// TwinCAT 3 PLC project PushcorpCtrl
// ProgramVersion: 3.1.4023.0
// libraries:
//   Tc2_Standard, * (Beckhoff Automation GmbH)
//   Tc2_System, * (Beckhoff Automation GmbH)
//   Tc3_EventLogger, * (Beckhoff Automation GmbH)
//   Tc3_Module, * (Beckhoff Automation GmbH)
//   BASIC,3.31,OSCAT
//   Util,3.5.11.0,System
// project tree:
//   DUTs/DoDi/IO/ ST_DoDi.TcDUT, ST_DoDi_in.TcDUT, ST_DoDi_out.TcDUT
//   DUTs/FCU/ E_FCU_ControlMode.TcDUT, ST_FcuControl.TcDUT, ST_FcuControl_in.TcDUT, ST_FcuControl_out.TcDUT
//   DUTs/FCU/IO/ ST_FCUFLEX.TcDUT, ST_FCUFLEX_in.TcDUT, ST_FCUFLEX_in_bits.TcDUT, ST_FCUFLEX_out.TcDUT
//   DUTs/Motoman/IO/ ST_MotomanIO.TcDUT, ST_MotomanIO_in.TcDUT, ST_MotomanIO_out.TcDUT
//   DUTs/Motoman/ ST_MotomanCtrl.TcDUT, ST_MotomanCtrl_in.TcDUT, ST_MotomanCtrl_out.TcDUT
//   DUTs/OPCUA/ ST_OpcuaStatus.TcDUT, ST_OpcuaStatusError.TcDUT, ST_OpcuaStatus_in.TcDUT, ST_OpcuaStatus_out.TcDUT, U_OpcuaError.TcDUT
//   DUTs/SPINDLE/IO/ ST_Spindle.TcDUT, ST_Spindle_in.TcDUT, ST_Spindle_in_bits.TcDUT, ST_Spindle_out.TcDUT, ST_Spindle_out_bits.TcDUT
//   DUTs/SPINDLE/ ST_SpindleControl.TcDUT, ST_SpindleControl_in.TcDUT, ST_SpindleControl_out.TcDUT
//   DUTs/Testing/ ST_TestBasicControl.TcDUT, ST_TestBasicControl_in.TcDUT, ST_TestBasicControl_out.TcDUT, ST_TestBasicControl_sub1.TcDUT
//   GVLs/ GVL_io.TcGVL, GVL_opcua.TcGVL
//   / PlcTask.TcTTO
//   POUs/ FB_FCU.TcPOU, FB_Motoman.TcPOU, FB_HeartbeatMonitor.TcPOU, FB_Spindle.TcPOU, FB_TestBasic.TcPOU, MAIN.TcPOU, prgMotoman.TcPOU, PRG_OpcuaMonitor.TcPOU
// real-time tasks:
//   TASK PlcTask: cycle T#1ms, priority 20, ADS port 350
//   TASK Task EthIp: cycle T#1ms, priority 1, ADS port 301
// I/O:
//   DEVICE Device 1 (EtherCAT), AmsNetId 192.168.125.39.2.1
//     Term 1 (EK1200) [EK1200-5000 EtherCAT Power supply (2A E-Bus)]
//       Term 2 (EL6070-0033) [EL6070-0033 1Ch. Licence key terminal, individual licences]
//       Term 3 (EL1008) [EL1008 8Ch. Dig. Input 24V, 3ms]
//       Term 4 (EL2008) [EL2008 8Ch. Dig. Output 24V, 0.5A]
//       Term 5 (EK1110) [EK1110 EtherCAT extension]
//   DEVICE Device 2 (TC3 EIP Scanner), AmsNetId 192.168.125.39.3.1
//     FCU (EtherNet/IP Slave (generic)) // <INFO> </INFO> <EDS> C:\TwinCAT\3.1\Config\Io\EtherNetIP\ </EDS>
//     Spindle (EtherNet/IP Slave (generic)) // <INFO> </INFO> <EDS> C:\TwinCAT\3.1\Config\Io\EtherNetIP\ </EDS>
//     DX200 EtherNet/IP(TM) Module // <INFO> 192.168.1.20, DX200 EtherNet/IP(TM) Module (ProdCode: 1281, Rev: 1.01, Mac: 00:26:73:d2:4a:d9) </INFO> <EDS> C:\TwinCAT\3.1\Config\Io\EtherNetIP\ </EDS>
// variable links:
//   PushcorpCtrl/PushcorpCtrl Instance <-> Device 1 (EtherCAT)/Term 1 (EK1200)/Term 3 (EL1008)
//     PlcTask Inputs/GVL_io.DI0 <-> Channel 1/GVL_io.DI0
//   PushcorpCtrl/PushcorpCtrl Instance <-> Device 1 (EtherCAT)/Term 1 (EK1200)/Term 4 (EL2008)
//     PlcTask Outputs/GVL_io.DO0 <-> Channel 1/GVL_io.DO0
//   PushcorpCtrl/PushcorpCtrl Instance <-> Device 2 (TC3 EIP Scanner)/DX200 EtherNet/IP(TM) Module
//     PlcTask Inputs/GVL_io.Motoman_Full.in/data <-> DX200 IO/Inputs/DX200_in
//     PlcTask Outputs/GVL_io.Motoman_Full.out <-> DX200 IO/Outputs/DX200_out
//   PushcorpCtrl/PushcorpCtrl Instance <-> Device 2 (TC3 EIP Scanner)/FCU (EtherNet/IP Slave (generic))
//     PlcTask Inputs/GVL_io.FCU_Full.DevState <-> Inputs/GVL_io.FCU_Full.DevState
//     PlcTask Inputs/GVL_io.FCU_Full.in <-> FCU IO/Inputs/GVL_io.FCU_Full.in
//     PlcTask Outputs/GVL_io.FCU_Full.out <-> FCU IO/Outputs/GVL_io.FCU_Full.out
//   PushcorpCtrl/PushcorpCtrl Instance <-> Device 2 (TC3 EIP Scanner)/Spindle (EtherNet/IP Slave (generic))
//     PlcTask Inputs/GVL_io.Spindle_Full.DevState <-> Inputs/GVL_io.Spindle_Full.DevState
//     PlcTask Inputs/GVL_io.Spindle_Full.in <-> Spindle IO/Inputs/GVL_io.Spindle_Full.in
//     PlcTask Outputs/GVL_io.Spindle_Full.out <-> Spindle IO/Outputs/GVL_io.Spindle_Full.out

CONFIGURATION PushcorpCtrl
    RESOURCE PLC ON TwinCAT3
        TASK PlcTask(INTERVAL := T#1ms, PRIORITY := 20);
        PROGRAM MAIN WITH PlcTask : MAIN;
    END_RESOURCE
END_CONFIGURATION

// ---- DUTs/DoDi/IO/ST_DoDi.TcDUT
TYPE ST_DoDi :
STRUCT	
	input	: ST_DoDi_in;	
	
	output	: ST_DoDi_out;	
END_STRUCT
END_TYPE

// ---- DUTs/DoDi/IO/ST_DoDi_in.TcDUT
TYPE ST_DoDi_in :
STRUCT
	DI0	AT %I*	: BOOL;
END_STRUCT
END_TYPE

// ---- DUTs/DoDi/IO/ST_DoDi_out.TcDUT
TYPE ST_DoDi_out :
STRUCT
	DO0	AT %Q*	: BOOL;
END_STRUCT
END_TYPE

// ---- DUTs/FCU/E_FCU_ControlMode.TcDUT
{attribute 'qualified_only'}
{attribute 'strict'}
TYPE E_FCU_ControlMode :
(
	Position := 0,
	Force := 1,
	SoftTouch := 3
) WORD;
END_TYPE

// ---- DUTs/FCU/IO/ST_FCUFLEX.TcDUT
{attribute 'pack_mode' := '2'}
TYPE ST_FCUFLEX :
STRUCT
	DevState AT %I* : UINT;
		
	in AT %I* : ST_FCUFLEX_in;
		
	out AT %Q* : ST_FCUFLEX_out;
END_STRUCT
END_TYPE

// ---- DUTs/FCU/IO/ST_FCUFLEX_in.TcDUT
{attribute 'pack_mode' := '2'}
TYPE ST_FCUFLEX_in :
STRUCT
	Flags : ST_FCUFLEX_in_bits;
	ActForce : INT;
	ActPos : WORD;
	AccelGravity : INT;
	CommandForce : INT;
	CommandPos : WORD;
	PayloadWeigth : WORD;
	ControlMode : WORD;
	MaxForce : WORD;
	MaxPos : WORD;
END_STRUCT
END_TYPE

// ---- DUTs/FCU/IO/ST_FCUFLEX_in_bits.TcDUT
TYPE ST_FCUFLEX_in_bits :
STRUCT
	hb : BIT;
	Hostcomm : BIT;
	ToolComm : BIT;
	MetricUnits : BIT;
	PosLimit : BIT;
	NegLimit : BIT;
	AtWeightPosition : BIT;
	WeighInProgress : BIT;
	WeightValid : BIT;
	 {attribute 'hide'}
	_reserved1 : BIT;
	 {attribute 'hide'}
	_reserved2 : BIT;
	 {attribute 'hide'}
	_reserved3 : BIT;
	 {attribute 'hide'}
	_reserved4 : BIT;
	 {attribute 'hide'}
	_reserved5 : BIT;
	 {attribute 'hide'}
	_reserved6 : BIT;
	 {attribute 'hide'}
	_reserved7 : BIT;
END_STRUCT
END_TYPE

// ---- DUTs/FCU/IO/ST_FCUFLEX_out.TcDUT
{attribute 'pack_mode' := '2'}
TYPE ST_FCUFLEX_out :
STRUCT
	CommandForce : INT;
	CommandPosition : WORD;
	PayloadWeight : WORD;
	ControlMode : WORD := 3;	// SoftTouch
	WeighPayloadNow : WORD;
END_STRUCT
END_TYPE

// ---- DUTs/FCU/ST_FcuControl.TcDUT
TYPE ST_FcuControl :
STRUCT
	status	: ST_OpcuaStatus;
	
	input	: ST_FcuControl_in;	
	
	{attribute 'OPC.UA.DA.Access' := '1'}
	output	: ST_FcuControl_out;
END_STRUCT
END_TYPE

// ---- DUTs/FCU/ST_FcuControl_in.TcDUT
{attribute 'OPC.UA.DA.StructuredType' := '1'}
TYPE ST_FcuControl_in :
STRUCT
	SetForce	: REAL;
	SetPosition	: REAL;
	SetWeight	: REAL;
	SetControlMode	: E_FCU_ControlMode := E_FCU_ControlMode.SoftTouch;
	WeighPayloadNow	: BOOL;
END_STRUCT
END_TYPE

// ---- DUTs/FCU/ST_FcuControl_out.TcDUT
{attribute 'OPC.UA.DA.StructuredType' := '1'}
TYPE ST_FcuControl_out :
STRUCT
	ActForce	: REAL;
	ActPos	: REAL;
	ActWeight	: REAL;
	Contact	: BOOL;
	WeightValid : BOOL;	
	Error	: UINT;
END_STRUCT
END_TYPE

// ---- DUTs/Motoman/IO/ST_MotomanIO.TcDUT
TYPE ST_MotomanIO :
STRUCT
	DevState AT %I* : UINT;
		
	in AT %I* : ST_MotomanIO_in;
		
	out AT %Q* : ST_MotomanIO_out;
END_STRUCT
END_TYPE

// ---- DUTs/Motoman/IO/ST_MotomanIO_in.TcDUT
TYPE ST_MotomanIO_in :
STRUCT
	data	: ARRAY[0..63] OF BYTE;
END_STRUCT
END_TYPE

// ---- DUTs/Motoman/IO/ST_MotomanIO_out.TcDUT
TYPE ST_MotomanIO_out :
STRUCT
	Cmd	: WORD;
	Vals	: ARRAY[0..5] OF WORD;
	Reserved	: ARRAY[0..49] OF BYTE;
END_STRUCT
END_TYPE

// ---- DUTs/Motoman/ST_MotomanCtrl.TcDUT
TYPE ST_MotomanCtrl :
STRUCT
	status	: ST_OpcuaStatus;
	
	input	: ST_MotomanCtrl_in;	
	
	{attribute 'OPC.UA.DA.Access' := '1'}
	output	: ST_MotomanCtrl_out;
END_STRUCT
END_TYPE

// ---- DUTs/Motoman/ST_MotomanCtrl_in.TcDUT
TYPE ST_MotomanCtrl_in :
STRUCT
	EnableJoystick	: BOOL;
	Value_1	: REAL;
	Value_2	: REAL;
	Value_3	: REAL;
	Value_4	: REAL;
	Value_5	: REAL;
	Value_6	: REAL;
END_STRUCT
END_TYPE

// ---- DUTs/Motoman/ST_MotomanCtrl_out.TcDUT
{attribute 'OPC.UA.DA.StructuredType' := '1'}
TYPE ST_MotomanCtrl_out :
STRUCT	
	Error	: UINT;
END_STRUCT
END_TYPE

// ---- DUTs/OPCUA/ST_OpcuaStatus.TcDUT
TYPE ST_OpcuaStatus :
STRUCT
	input	: ST_OpcuaStatus_in;
	
	{attribute 'OPC.UA.DA.Access' := '1'}
	output	: ST_OpcuaStatus_out;
END_STRUCT
END_TYPE

// ---- DUTs/OPCUA/ST_OpcuaStatusError.TcDUT
TYPE ST_OpcuaStatusError :
STRUCT
	DevDisconnected	: BIT;
	ClientHbLost	: BIT;
END_STRUCT
END_TYPE

// ---- DUTs/OPCUA/ST_OpcuaStatus_in.TcDUT
TYPE ST_OpcuaStatus_in :
STRUCT
	Heartbeat	: BOOL;
END_STRUCT
END_TYPE

// ---- DUTs/OPCUA/ST_OpcuaStatus_out.TcDUT
TYPE ST_OpcuaStatus_out :
STRUCT
	Heartbeat	: BOOL;
	Error	: UINT;	// 0 = No error
	Connected	: BOOL;
END_STRUCT
END_TYPE

// ---- DUTs/OPCUA/U_OpcuaError.TcDUT
TYPE U_OpcuaError :
UNION
	Value	: UINT;
	Bits	: ST_OpcuaStatusError;
END_UNION
END_TYPE

// ---- DUTs/SPINDLE/IO/ST_Spindle.TcDUT
{attribute 'pack_mode' := '2'}
TYPE ST_Spindle :
STRUCT
	DevState AT %I*	: UINT;
	in AT %I*	: ST_Spindle_in;
	out	 AT %Q* : ST_Spindle_out;
END_STRUCT
END_TYPE

// ---- DUTs/SPINDLE/IO/ST_Spindle_in.TcDUT
TYPE ST_Spindle_in :
STRUCT
	flags	: ST_Spindle_in_bits;
	SpindleSpeed	: INT;
	MotorLoad	: INT;
END_STRUCT
END_TYPE

// ---- DUTs/SPINDLE/IO/ST_Spindle_in_bits.TcDUT
{attribute 'pack_mode' := '2'}
TYPE ST_Spindle_in_bits :
STRUCT
	Contactor1	: BIT;
	Contactor2	: BIT;
	DriveError	: BIT;
	RpmLT5		: BIT;	
	DI5			: BIT;
	DI6			: BIT;
	DI7			: BIT;
	DI8			: BIT;
	Reserved	: BIT;	// Force 2 bytes, probably not needed
END_STRUCT
END_TYPE

// ---- DUTs/SPINDLE/IO/ST_Spindle_out.TcDUT
TYPE ST_Spindle_out :
STRUCT
	flags	: ST_Spindle_out_bits;
	SpindleSpeed	: INT;
	Reserved	: INT;
END_STRUCT
END_TYPE

// ---- DUTs/SPINDLE/IO/ST_Spindle_out_bits.TcDUT
{attribute 'pack_mode' := '2'}
TYPE ST_Spindle_out_bits :
STRUCT
	ServoEnable	: BIT;
	ResetFault	: BIT;
	DO3	: BIT;
	DO4	: BIT;
	DO5	: BIT;
	DO6	: BIT;
	DO7	: BIT;
	DO8	: BIT;	
	Reserved	: BIT;	// Force 2 bytes, probably not needed
END_STRUCT
END_TYPE

// ---- DUTs/SPINDLE/ST_SpindleControl.TcDUT
{attribute 'OPC.UA.DA.StructuredType' := '1'}
TYPE ST_SpindleControl :
STRUCT
	status	: ST_OpcuaStatus;
	
	input	: ST_SpindleControl_in;
	
	{attribute 'OPC.UA.DA.Access' := '1'}
	output	: ST_SpindleControl_out;
END_STRUCT
END_TYPE

// ---- DUTs/SPINDLE/ST_SpindleControl_in.TcDUT
{attribute 'OPC.UA.DA.StructuredType' := '1'}
TYPE ST_SpindleControl_in :
STRUCT
	Execute	: BOOL;
	(*{attribute 'OPC.UA.DA.AnalogItemType' := '1'}
	{attribute 'OPC.UA.DA.AnalogItemType.EngineeringUnits' := '5059638'}
	{attribute 'OPC.UA.DA.AnalogItemType.EURange' := '-15000.0:15000.0'}
	{attribute 'OPC.UA.DA.AnalogItemType.WriteBehavior' := '1'}*)
	SetVelo	: REAL;
END_STRUCT
END_TYPE

// ---- DUTs/SPINDLE/ST_SpindleControl_out.TcDUT

TYPE ST_SpindleControl_out :
STRUCT
	ActVelo	: REAL;	//Speed in RPMs
	Ready	: BOOL;
	Error	: UINT;	// 0 = No error
END_STRUCT
END_TYPE

// ---- DUTs/Testing/ST_TestBasicControl.TcDUT
TYPE ST_TestBasicControl :
STRUCT
	status	: ST_OpcuaStatus;	
	input	: ST_TestBasicControl_in;	
	
	{attribute 'OPC.UA.DA.Access' := '1'}
	output	: ST_TestBasicControl_out;
END_STRUCT
END_TYPE

// ---- DUTs/Testing/ST_TestBasicControl_in.TcDUT
TYPE ST_TestBasicControl_in :
STRUCT
	arrTest	: ARRAY[0..10] OF DINT;
	DO0	: BOOL;
	in1	: DINT;
	int2	: DINT;
	stSub1In	: ST_TestBasicControl_sub1; 
	inStr1	: STRING(255);	
END_STRUCT
END_TYPE

// ---- DUTs/Testing/ST_TestBasicControl_out.TcDUT
TYPE ST_TestBasicControl_out :
STRUCT
	DI0	: BOOL;
	out1	: DINT;
	out2	: DINT;
	stSub1Out	: ST_TestBasicControl_sub1;
	outStr1	: STRING(255);
	arrTest	: ARRAY[0..1] OF BYTE;
END_STRUCT
END_TYPE

// ---- DUTs/Testing/ST_TestBasicControl_sub1.TcDUT
TYPE ST_TestBasicControl_sub1 :
STRUCT
	sub1val	: DINT;
END_STRUCT
END_TYPE

// ---- GVLs/GVL_io.TcGVL
{attribute 'qualified_only'}
VAR_GLOBAL
	DI0 AT %I*	: BOOL;
	DO0 AT %Q*	: BOOL;
	
	Spindle_Full	: ST_Spindle;
	FCU_Full	: ST_FCUFLEX;
	
	
	DX200_in AT %I*	: ARRAY [0..7] OF BYTE;
	DX200_out AT %Q*	: ARRAY [0..7] OF BYTE;
	
	Motoman_Full	: ST_MotomanIO;
END_VAR

// ---- GVLs/GVL_opcua.TcGVL
{attribute 'qualified_only'}
VAR_GLOBAL
	{attribute 'OPC.UA.DA' := '1'}	
	stFcuControl	: ST_FcuControl;
	
	{attribute 'OPC.UA.DA' := '1'}
	stSpindleControl	: ST_SpindleControl;
	
	{attribute 'OPC.UA.DA' := '1'}	
	stTestBasic	: ST_TestBasicControl;
	
	{attribute 'OPC.UA.DA' := '1'}	
	stMotomanControl	: ST_MotomanCtrl;
END_VAR

// ---- POUs/MAIN.TcPOU
PROGRAM MAIN
VAR
	fbSpindle	: FB_Spindle;
	fbFcu	: FB_FCU;
	fbMotoman	: FB_Motoman;
	
	
	spin: REFERENCE TO ST_SpindleControl;
	fcu: REFERENCE TO ST_FcuControl;
	
	motoman	: REFERENCE TO ST_MotomanCtrl;
	motomanErr: BOOL;
END_VAR

//prgMotoman();

// Set ref vars for convenience of shorter names 
spin REF= GVL_opcua.stSpindleControl;
fcu REF=GVL_opcua.stFcuControl;
motoman REF= GVL_opcua.stMotomanControl;

// Monitor opcua heartbeat data in a Method for convenience.  This can be easily ignored if calling the FB without opcua 
fbSpindle.OpcuaMonitor(OpcuaData:= spin, Error=> );
fbSpindle(
	Enable:= spin.input.Execute, 
	SetVelo:= spin.input.SetVelo, 
	data:= GVL_io.Spindle_Full, 
	ActVelo=> spin.output.ActVelo, 
	Ready=> spin.output.Ready, 
	Error=> spin.output.Error);


fbFcu.OpcuaMonitor(OpcuaData:= fcu, Error=> );
fbFcu(
	SetForce:= fcu.input.SetForce, 
	SetPosition:= fcu.input.SetPosition, 
	SetWeight:= fcu.input.SetWeight, 
	SetControlMode:= fcu.input.SetControlMode, 
	WeightPayload:= fcu.input.WeighPayloadNow, 
	data:= gvl_io.FCU_Full, 
	ActForce=> fcu.output.ActForce, 
	ActPos=> fcu.output.ActPos, 
	ActWeight=> fcu.output.ActWeight,
	Contact=> fcu.output.Contact,
	WeightValid=> fcu.output.WeightValid, 
	Error=> fcu.output.Error);
	
fbMotoman.OpcuaMonitor(OpcuaData:= GVL_opcua.stMotomanControl, Error=> motomanErr);
fbMotoman(
	EnableJoystick:= NOT motomanErr, 
	Value_1:= motoman.input.Value_1, 
	Value_2:= motoman.input.Value_2, 
	Value_3:= motoman.input.Value_3, 
	Value_4:= , 
	Value_5:= , 
	Value_6:= , 
	data:= GVL_io.Motoman_Full, 
	Error=> );
	
// DI0 := DO0, for testing
GVL_io.DO0 := GVL_opcua.stTestBasic.input.DO0;
GVL_opcua.stTestBasic.output.DI0 := GVL_io.DI0;

END_PROGRAM

// ---- POUs/FB_Spindle.TcPOU
FUNCTION_BLOCK FB_Spindle
VAR_INPUT
	Enable	: BOOL; // Enable the servo
	SetVelo	: REAL;	// Speed in RPMs
END_VAR
VAR_IN_OUT
	data	: ST_Spindle;	// Ethernet IP data
END_VAR
VAR_OUTPUT
	ActVelo	: REAL;	//Speed in RPMs
	Ready	: BOOL; // Servo ready to move
	Error	: UINT; // 0 = OK, 1 = not connected
END_VAR
VAR
	rTargetVel	: REAL;	
	fbTrigEnable	: BOOL;	
	iState	: DINT;	
	fbDelay	: TON;
	bRunDelay	: BOOL;
	uiDevState: UINT;
END_VAR

IF NOT Enable THEN
	iState := 0;
END_IF

uiDevState := data.DevState;

// Scale target rpm
rTargetVel := SCALE_R(
				X:= SetVelo, 
				I_LO:= -15000, 
				I_HI:= 15000, 
				O_LO:= -30000, 
				O_HI:= 30000);
				
fbDelay(IN:= bRunDelay, PT:= T#1000MS, Q=> , ET=> );				

CASE iState OF
0:	// Default, set all output to 0
	MEMSET(ADR(data.out.flags), 0, SIZEOF(data.out.flags));
	bRunDelay := FALSE;
	IF Enable THEN
		iState := 10;
	END_IF
10:
	IF data.in.flags.DriveError THEN
		data.out.flags.ResetFault := TRUE;
		iState := 20;	// Reset state
	ELSE			
		iState := 100;	// OK to run
	END_IF	
20:
	data.out.flags.ServoEnable := FALSE;
	data.out.flags.ResetFault := data.in.flags.DriveError;
	bRunDelay := TRUE;	// Don't try to power on for at least a second
	IF NOT data.in.flags.DriveError AND fbDelay.Q THEN
		iState := 100;
		bRunDelay := FALSE;
	END_IF
	
100:
	data.out.flags.ServoEnable := TRUE;
	data.out.SpindleSpeed := TO_INT(rTargetVel);
	
	IF data.in.flags.DriveError THEN
		iState := 999;
	END_IF
	
999: // Stay in fault state until error can be examined
	data.out.flags.ServoEnable := FALSE;
	;
END_CASE


Error := TO_UINT(data.in.flags.DriveError);
Ready := Error = 0 AND data.in.flags.Contactor1 AND data.in.flags.Contactor2 AND data.DevState = 0;


IF data.in.flags.RpmLT5 THEN
	ActVelo := 0;
ELSE
	ActVelo := SCALE_R(
		X:= data.in.SpindleSpeed, 
		I_LO:= -30000, 
		I_HI:= 30000, 
		O_LO:= -15000, 
		O_HI:= 15000);
END_IF

METHOD OpcuaMonitor : BOOL
VAR_INPUT
END_VAR
VAR_IN_OUT
	OpcuaData	: ST_SpindleControl;
END_VAR
VAR_OUTPUT
	Error	: BOOL;
END_VAR
VAR_INST
	fbHbMonitor	: FB_HeartbeatMonitor;
	fbBlink	: BLINK;
END_VAR
fbHbMonitor(IN:= OpcuaData.status.input.Heartbeat, PT:= T#2.5S, Q=> );

IF NOT fbHbMonitor.Q THEN
	MEMSET(ADR(OpcuaData.input), 0, SIZEOF(OpcuaData.input));
	Error := TRUE;
ELSE
	Error := FALSE;
END_IF

fbBlink(ENABLE:= TRUE, TIMELOW:= T#500MS, TIMEHIGH:= T#500MS, OUT=> OpcuaData.status.output.Heartbeat);
OpcuaData.status.output.Connected := (THIS^.uiDevState = 0);
END_METHOD

END_FUNCTION_BLOCK

// ---- POUs/FB_HeartbeatMonitor.TcPOU
FUNCTION_BLOCK FB_HeartbeatMonitor
VAR_INPUT
	IN	: BOOL;
	PT	: TIME := T#2S;
END_VAR
VAR_OUTPUT
	Q	: BOOL;
END_VAR
VAR
	fbHbTimeout: TON;
	bLastHB: BOOL;
END_VAR

fbHbTimeout(IN:= (bLastHB = IN), PT:= PT, Q=> Q, ET=> );
Q := NOT fbHbTimeout.Q;
bLastHB := IN;

END_FUNCTION_BLOCK

// ---- POUs/FB_FCU.TcPOU
FUNCTION_BLOCK FB_FCU
VAR_INPUT
	SetForce	: REAL;	// Desired force in NM
	SetPosition	: REAL;	// Desired position in mm
	SetWeight	: REAL;	// Manually specify the weight, leave 0 if using WeightPayload
	SetControlMode	: E_FCU_ControlMode := E_FCU_ControlMode.Force;	// Position, Force, Soft Touch
	WeightPayload	: BOOL;	// Weight the payload now
END_VAR
VAR_IN_OUT
	data	: ST_FCUFLEX;	// Raw data from Ethernet/IP
END_VAR
VAR_OUTPUT
	ActForce	: REAL;	// Actual force in NM
	ActPos	: REAL;	// Actual position in mm
	ActWeight	: REAL;	// Actual weight in KG
	Contact	: BOOL;	// Contact state
	WeightValid : BOOL; // Is the weight valid or not initialized
	Error	: UINT;	// 
END_VAR
VAR
	bLastHB	: BOOL;
	bOk	: BOOL;	
	fbHbTimeout	: TON;
	
	rScaledForce: REAL;
	rTemp	: REAL;	
	rMaxPos	: REAL;
	uiDevState: UINT;
END_VAR

uiDevState := data.DevState;
// Check comms and heartbeat
bOk := TRUE;	
fbHbTimeout(IN:= (bLastHB = data.in.Flags.hb), PT:= T#2S, Q=> , ET=> );
bLastHB := data.in.Flags.hb;
	
IF fbHbTimeout.Q OR NOT data.in.Flags.Hostcomm OR NOT data.in.Flags.ToolComm THEN
	bOk := FALSE;
END_IF

// Scale data from FCU
ActForce := data.in.ActForce / 10.0;
ActPos := data.in.ActPos / 100.0;
ActWeight := data.in.PayloadWeigth / 100.0;
// Determine contact
rMaxPos := data.in.MaxPos  / 100.0;
Contact := (ActPos >= 2.0 AND ActPos <= rMaxPos - 2.0);
WeightValid := data.in.Flags.WeightValid;

// Scale and write data to FCU
data.out.ControlMode := TO_WORD(SetControlMode);
data.out.CommandForce := TO_INT(SetForce * 10.0);
data.out.CommandPosition := TO_WORD(SetPosition * 100.0);
data.out.PayloadWeight := TO_WORD(SetWeight * 100.0);
data.out.WeighPayloadNow := TO_WORD(WeightPayload);



Error := TO_UINT(NOT bOk);

METHOD OpcuaMonitor : BOOL
VAR_INPUT
END_VAR
VAR_IN_OUT
	OpcuaData	: ST_FcuControl;
END_VAR
VAR_OUTPUT
	Error	: BOOL;
END_VAR
VAR_INST
	fbHbMonitor	: FB_HeartbeatMonitor;
	fbBlink	: BLINK;	
	err	: U_OpcuaError;
END_VAR
fbHbMonitor(IN:= OpcuaData.status.input.Heartbeat, PT:= T#2.5S, Q=> );
err.Value := 0;
IF NOT fbHbMonitor.Q THEN
	// There's no way to simply disable the fcu and it defaults to position mode.  Trying to move to position 0
	// will cause a significant force
	OpcuaData.input.SetControlMode := E_FCU_ControlMode.SoftTouch;
	OpcuaData.input.SetForce := 0;
	OpcuaData.input.WeighPayloadNow := FALSE;
	
	err.Bits.ClientHbLost := TRUE;
END_IF

OpcuaData.status.output.Connected := (THIS^.uiDevState = 0);
IF NOT OpcuaData.status.output.Connected THEN	// higher priority
	err.Bits.DevDisconnected := TRUE;	
END_IF

Error := err.Value <> 0;
OpcuaData.status.output.Error := err.Value;

fbBlink(ENABLE:= TRUE, TIMELOW:= T#500MS, TIMEHIGH:= T#500MS, OUT=> OpcuaData.status.output.Heartbeat);
END_METHOD

END_FUNCTION_BLOCK

// ---- POUs/FB_Motoman.TcPOU
FUNCTION_BLOCK FB_Motoman
VAR_INPUT
	EnableJoystick	: BOOL;
	Value_1	: REAL;
	Value_2	: REAL;
	Value_3	: REAL;
	Value_4	: REAL;
	Value_5	: REAL;
	Value_6	: REAL;	
END_VAR
VAR_IN_OUT
	data	: ST_MotomanIO;	// Raw data from Ethernet/IP
END_VAR
VAR_OUTPUT	
	Error	: UINT;	// 
END_VAR
VAR
	uiDevState: UINT;
	bOk	: BOOL;	
	fbHbTimeout	: TON;
	
	rMaxOutVel : REAL := 1000;

	
	
	pInt	: POINTER TO INT;
	pWord	: POINTER TO WORD;
END_VAR

uiDevState := data.DevState;
// Check comms and heartbeat
bOk := TRUE;	


(*valTemp := LIMIT(-0.6, Value_1, 0.6);

tempLin := F_LIN2(
	X:= valTemp, 
	X1:= -0.6, 
	Y1:= -1000, 
	X2:= 0.6, 
	Y2:= 1000);
	
tempInt := TO_INT(tempLin);

MEMMOVE(ADR(data.out.Vals[0]), ADR(tempInt), 2);
//data.out.Vals[0] := tempInt;
*)

data.out.Vals[0] := PrepareValue(Value_1, rMaxOutVel);
data.out.Vals[1] := PrepareValue(Value_2, rMaxOutVel);
data.out.Vals[2] := PrepareValue(Value_3, rMaxOutVel);

data.out.Cmd.0 := EnableJoystick;

data.out.Cmd.1 := data.out.Vals[0] <> 0 OR data.out.Vals[1] <> 0 OR data.out.Vals[2] <> 0;

IF NOT EnableJoystick THEN 
	MEMSET(ADR(data.out.Cmd), 0, SIZEOF(data.out.Cmd));
	MEMSET(ADR(data.out.Vals), 0, SIZEOF(data.out.Vals));
END_IF
Error := TO_UINT(NOT bOk);

METHOD OpcuaMonitor : BOOL
VAR_INPUT
END_VAR
VAR_IN_OUT
	OpcuaData	: ST_MotomanCtrl;
END_VAR
VAR_OUTPUT
	Error	: BOOL;
END_VAR
VAR_INST
	fbHbMonitor	: FB_HeartbeatMonitor;
	fbBlink	: BLINK;	
	err	: U_OpcuaError;
END_VAR
fbHbMonitor(IN:= OpcuaData.status.input.Heartbeat, PT:= T#2.5S, Q=> );

IF NOT fbHbMonitor.Q THEN
	MEMSET(ADR(OpcuaData.input), 0, SIZEOF(OpcuaData.input));
	Error := TRUE;
ELSE
	Error := FALSE;
END_IF

fbBlink(ENABLE:= TRUE, TIMELOW:= T#500MS, TIMEHIGH:= T#500MS, OUT=> OpcuaData.status.output.Heartbeat);
OpcuaData.status.output.Connected := (THIS^.uiDevState = 0);
END_METHOD

METHOD PrepareValue : INT
VAR_INPUT
	SetVal	: REAL;
	MaxOut	: REAL := 1000;
END_VAR
VAR
	tempWord: WORD;
	tempInt	: INT;
	valTemp: REAL;
	tempLin: REAL;
END_VAR
valTemp := LIMIT(-0.6, SetVal, 0.6);

tempLin := F_LIN2(
	X:= valTemp, 
	X1:= -0.6, 
	Y1:= -MaxOut, 
	X2:= 0.6, 
	Y2:= MaxOut);
	
tempInt := TO_INT(tempLin);

MEMMOVE(ADR(PrepareValue), ADR(tempInt), 2);
END_METHOD

END_FUNCTION_BLOCK

// ---- POUs/FB_TestBasic.TcPOU
FUNCTION_BLOCK FB_TestBasic
VAR_INPUT
	DO0	: BOOL; // Enable the servo	
END_VAR
VAR_IN_OUT
	data	: ST_TestBasic;	// Ethernet IP data
END_VAR
VAR_OUTPUT
	DI0	: BOOL;
	Ready	: BOOL;
	Error	: UINT; 
END_VAR
VAR
END_VAR

METHOD OpcuaMonitor : BOOL
VAR_INPUT
END_VAR
VAR_IN_OUT
	Data	: ST_SpindleControl;
END_VAR
VAR_OUTPUT
	Error	: BOOL;
END_VAR
VAR_INST
	fbHbMonitor	: FB_HeartbeatMonitor;
END_VAR
fbHbMonitor(IN:= Data.status.input.Heartbeat, PT:= T#2.5S, Q=> );

IF NOT fbHbMonitor.Q THEN
	MEMSET(ADR(Data.input), 0, SIZEOF(Data.input));
	Error := TRUE;
ELSE
	Error := FALSE;
END_IF
END_METHOD

END_FUNCTION_BLOCK

// ---- POUs/prgMotoman.TcPOU
PROGRAM prgMotoman
VAR
	pReal	: POINTER TO REAL;
	rVal	: REAL;
	
	pInt	: POINTER TO INT;
	iVal	: INT;
	
	fbsin	: BASIC.GEN_SIN;
	rSinOut: REAL;
	
	pRun	: POINTER TO BOOL;
	bRun	: BOOL;
	
	bUpdate: BOOL;
	
	bRunning : BOOL;
	
	fbTimer	: TOF;
	
	iCycles	: DINT;
END_VAR

pReal := ADR(GVL_io.DX200_out[0]);
//pReal^ := rVal;

pInt := ADR(GVL_io.DX200_out[4]);
//pInt^ := iVal;

pRun := ADR(GVL_io.DX200_out[0]);
pRun^ := bRun;

bRunning := GVL_io.DX200_in[0].0;

fbsin(
	PT:= T#5S, 
	AM:= 2000, 
	OS:= , 
	DL:= , 
	Q=> , 
	Out=> rSinOut);
	
IF rSinOut >= 100 THEN
	rSinOut := 100;
ELSIF rSinOut <= -100 THEN
	rSinOut := -100;
END_IF
	
IF bUpdate THEN
	pInt^ := TO_INT(rSinOut);
	iCycles := 0;
ELSE
	bRun := FALSE;
	pInt^ := 0;	
	IF bRunning THEN
		iCycles := iCycles + 1;
	END_IF
END_IF

END_PROGRAM

// ---- POUs/PRG_OpcuaMonitor.TcPOU
PROGRAM PRG_OpcuaMonitor

VAR_OUTPUT
	Error : BOOL;	
END_VAR
VAR
	fbFCUHb	: FB_HeartbeatMonitor;
	fbSpindleHb	: FB_HeartbeatMonitor;
END_VAR

Error := FALSE;

fbFCUHb(IN:= GVL_opcua.stFcuControl.status.input.Heartbeat, T:= T#2.5S, Q=> );
IF NOT fbFCUHb.Q THEN
	// There's no way to simply disable the fcu.  
	GVL_opcua.stFcuControl.input.SetControlMode := E_FCU_ControlMode.SoftTouch;
	GVL_opcua.stFcuControl.input.SetForce := 0;	
	Error := TRUE;
ELSE
	Error := FALSE;
END_IF



fbSpindleHb(IN:= GVL_opcua.stSpindleControl.status.input.Heartbeat, T:= T#2.5S, Q=> );
IF NOT fbSpindleHb.Q THEN
	MEMSET(ADR(GVL_opcua.stSpindleControl.input), 0, SIZEOF(GVL_opcua.stSpindleControl.input));
	Error := TRUE;
ELSE
	Error := FALSE;
END_IF

END_PROGRAM
